(*udt (user defined type) of Beckhoff EK1100 - EtherCAT Bus Coupler (Slave):
	auth. Brent Lekx-Toniolo of Toniolo Research & Development Inc.; 
	July 2010; version 1.0*)


TYPE udt_EK1100 :
STRUCT
 	InfoData: udt_ECATSlave_Status;
END_STRUCT
END_TYPE

(* stored: Version 1.1.0.1, ProductVersion 3.1.4024.9
   DUT udt_EK1100: Id {8fb6fcd6-0651-4267-a78f-d1b2a5558d77} *)
